FUNCTION_BLOCK FB_LevitationSystem IMPLEMENTS ITF_HighLevelSystem
VAR_INPUT
	eState : LevitationSystemSTM;
	nTGControlOption : USINT;
	eActivationStatus : ActivationStatus;
END_VAR
VAR_OUTPUT
	bEnableCurrentController : BOOL;
	bEnableIControl : BOOL;
	bEnablePControl : BOOL;
END_VAR
VAR
	fbEqualizingControl			: FB_EqualizingController;
	fbTrajectoryGeneratorXMC1	: FB_TrajectoryGenerator;
	fbTrajectoryGeneratorXMC2	: FB_TrajectoryGenerator;
	fbTrajectoryGeneratorXMC3	: FB_TrajectoryGenerator;
	fbTrajectoryGeneratorXMC4	: FB_TrajectoryGenerator;
	
	fActualLevDistanceForFmag : ARRAY [0..3] OF REAL;
	fActualLevCurrentForFmag : ARRAY [0..3] OF REAL;
END_VAR

IF eActivationStatus = ActivationStatus.Enabled THEN
	//High Level State Machine
	CASE eState OF
		LevitationSystemSTM.Idling:
			;
			
			
		LevitationSystemSTM.Stationary:
			bEnableCurrentController := FALSE;
			fbTrajectoryGeneratorXMC1.bTransition := FALSE;
			fbTrajectoryGeneratorXMC2.bTransition := FALSE;
			fbTrajectoryGeneratorXMC3.bTransition := FALSE;
			fbTrajectoryGeneratorXMC4.bTransition := FALSE;

			fbEqualizingControl.bActive := FALSE;		
		
			doSetOperationMode();
			
			fbTrajectoryGeneratorXMC1();
			fbTrajectoryGeneratorXMC2();
			fbTrajectoryGeneratorXMC3();
			fbTrajectoryGeneratorXMC4();
			fbEqualizingControl();
			
		LevitationSystemSTM.Transitioning:
			bEnableCurrentController := TRUE;
			fbTrajectoryGeneratorXMC1.bTransition := TRUE;
			fbTrajectoryGeneratorXMC2.bTransition := TRUE;
			fbTrajectoryGeneratorXMC3.bTransition := TRUE;
			fbTrajectoryGeneratorXMC4.bTransition := TRUE;
			
			fbEqualizingControl.bActive := FALSE;
			
			fbTrajectoryGeneratorXMC1();
			fbTrajectoryGeneratorXMC2();
			fbTrajectoryGeneratorXMC3();
			fbTrajectoryGeneratorXMC4();
			fbEqualizingControl();
			
			
		LevitationSystemSTM.HoldingAirGap:
			bEnableCurrentController := FALSE;
			fbTrajectoryGeneratorXMC1.bTransition := FALSE;
			fbTrajectoryGeneratorXMC2.bTransition := FALSE;
			fbTrajectoryGeneratorXMC3.bTransition := FALSE;
			fbTrajectoryGeneratorXMC4.bTransition := FALSE;
			
			fbEqualizingControl.bActive := TRUE;
			
			doCalculateFmagValuesForEC(	fActualLevDistance := fActualLevDistanceForFmag,			//to be implemented
										fActualCurrent := fActualLevCurrentForFmag);
			
			fbTrajectoryGeneratorXMC1();
			fbTrajectoryGeneratorXMC2();
			fbTrajectoryGeneratorXMC3();
			fbTrajectoryGeneratorXMC4();
			fbEqualizingControl();
			
			
		LevitationSystemSTM.TransitioningToZero:
			bEnableCurrentController := TRUE;
			fbTrajectoryGeneratorXMC1.bTransition := TRUE;
			fbTrajectoryGeneratorXMC2.bTransition := TRUE;
			fbTrajectoryGeneratorXMC3.bTransition := TRUE;
			fbTrajectoryGeneratorXMC4.bTransition := TRUE;
			
			fbEqualizingControl.bActive := FALSE;
			
			doSetPresetTGValuesForBackToGround();		//to be implemented with Controller structure
			
			fbTrajectoryGeneratorXMC1();
			fbTrajectoryGeneratorXMC2();
			fbTrajectoryGeneratorXMC3();
			fbTrajectoryGeneratorXMC4();
			fbEqualizingControl();
			
	END_CASE	

END_IF

PROPERTY PUBLIC aECOutputZVector : ARRAY [0..3] OF REAL
GET
END_GET
END_PROPERTY

PROPERTY PUBLIC aTGActualLevAcceleration : ARRAY [0..3] OF REAL
SET
END_SET
END_PROPERTY

PROPERTY PUBLIC aTGActualLevCurrent : ARRAY [0..3] OF REAL
SET
fActualLevCurrentForFmag := aTGActualLevCurrent;
END_SET
END_PROPERTY

PROPERTY PUBLIC aTGActualLevDistance : ARRAY [0..3] OF REAL
SET
fActualLevDistanceForFmag := aTGActualLevDistance;
END_SET
END_PROPERTY

PROPERTY PUBLIC aTGActualLevVelocity : ARRAY [0..3] OF REAL
SET
END_SET
END_PROPERTY

PROPERTY PUBLIC aTGOutputLevAcceleration : ARRAY [0..3] OF REAL
GET
END_GET
END_PROPERTY

PROPERTY PUBLIC aTGOutputLevCurrent : ARRAY [0..3] OF REAL
GET
END_GET
END_PROPERTY

PROPERTY PUBLIC aTGOutputLevDistance : ARRAY [0..3] OF REAL
GET
END_GET
END_PROPERTY

PROPERTY PUBLIC aTGOutputLevForce : ARRAY [0..3] OF REAL
GET
END_GET
END_PROPERTY

PROPERTY PUBLIC aTGOutputLevVelocity : ARRAY [0..3] OF REAL
GET
END_GET
END_PROPERTY

PROPERTY PUBLIC aTGOutputLevVoltage : ARRAY [0..3] OF REAL
GET
END_GET
END_PROPERTY

PROPERTY PUBLIC bTrajectoryCompleted : BOOL
GET
VAR
	bTrajectoryCompletedXMC1 : BOOL;
	bTrajectoryCompletedXMC2 : BOOL;
	bTrajectoryCompletedXMC3 : BOOL;
	bTrajectoryCompletedXMC4 : BOOL;
END_VAR
bTrajectoryCompletedXMC1 := fbTrajectoryGeneratorXMC1.bTrajectoryCompleted;
bTrajectoryCompletedXMC2 := fbTrajectoryGeneratorXMC2.bTrajectoryCompleted;
bTrajectoryCompletedXMC3 := fbTrajectoryGeneratorXMC3.bTrajectoryCompleted;
bTrajectoryCompletedXMC4 := fbTrajectoryGeneratorXMC4.bTrajectoryCompleted;

IF bTrajectoryCompletedXMC1 AND bTrajectoryCompletedXMC2 AND bTrajectoryCompletedXMC3 AND bTrajectoryCompletedXMC4 THEN
	bTrajectoryCompleted := TRUE;
ELSE
	bTrajectoryCompleted := FALSE;
END_IF
END_GET
SET
END_SET
END_PROPERTY

METHOD PRIVATE doCalculateFmagValuesForEC
VAR_INPUT
	fActualLevDistance : ARRAY [0..3] OF REAL;
	fActualCurrent		: ARRAY [0..3] OF REAL;
END_VAR
fbEqualizingControl.fActualDeltaFmag := 0;
END_METHOD

METHOD PRIVATE doSetOperationMode
VAR_INPUT
END_VAR
IF nTGControlOption.0 THEN
	fbTrajectoryGeneratorXMC1.eMode := TGControllerMode.IControl;
	fbTrajectoryGeneratorXMC2.eMode := TGControllerMode.IControl;
	fbTrajectoryGeneratorXMC3.eMode := TGControllerMode.IControl;
	fbTrajectoryGeneratorXMC4.eMode := TGControllerMode.IControl;
	
	bEnableIControl := TRUE;
	bEnablePControl := FALSE;
END_IF

IF nTGControlOption.1 THEN
	fbTrajectoryGeneratorXMC1.eMode := TGControllerMode.PControl;
	fbTrajectoryGeneratorXMC2.eMode := TGControllerMode.PControl;
	fbTrajectoryGeneratorXMC3.eMode := TGControllerMode.PControl;
	fbTrajectoryGeneratorXMC4.eMode := TGControllerMode.PControl;
	
	bEnableIControl := FALSE;
	bEnablePControl := TRUE;
END_IF
END_METHOD

METHOD PRIVATE doSetPresetTGValuesForBackToGround
VAR_INPUT
END_VAR
END_METHOD

PROPERTY eCondition : HighLevelCondition
GET
IF eActivationStatus = ActivationStatus.Disabled THEN
	eCondition := HighLevelCondition.SLEEP;
ELSE
	IF fbTrajectoryGeneratorXMC1.eCondition = SubLevelCondition.RUN AND fbTrajectoryGeneratorXMC2.eCondition = SubLevelCondition.RUN AND fbTrajectoryGeneratorXMC3.eCondition = SubLevelCondition.RUN AND fbTrajectoryGeneratorXMC4.eCondition = SubLevelCondition.RUN AND fbEqualizingControl.eCondition = SubLevelCondition.RUN THEN
		eCondition := HighLevelCondition.RUN;
	ELSE
		eCondition := HighLevelCondition.INIT;
	END_IF
END_IF
END_GET
END_PROPERTY

PROPERTY PUBLIC fTGDesiredLevAcceleration : REAL
SET
END_SET
END_PROPERTY

PROPERTY PUBLIC fTGDesiredLevDistance : REAL
SET
END_SET
END_PROPERTY

PROPERTY PUBLIC fTGDesiredLevTime : REAL
SET
END_SET
END_PROPERTY

PROPERTY PUBLIC fTGDesiredLevVelocity : REAL
SET
END_SET
END_PROPERTY

PROPERTY nErrorID : UDINT
GET
VAR
	nErrorBitsTG1 : UDINT;
	nErrorBitsTG2 : UDINT;
	nErrorBitsTG3 : UDINT;
	nErrorBitsTG4 : UDINT;
	nErrorBitsEC	: UDINT;
END_VAR
nErrorBitsTG1 := fbTrajectoryGeneratorXMC1.nErrorID;
nErrorBitsTG2 := fbTrajectoryGeneratorXMC2.nErrorID;
nErrorBitsTG3 := fbTrajectoryGeneratorXMC3.nErrorID;
nErrorBitsTG4 := fbTrajectoryGeneratorXMC4.nErrorID;
nErrorBitsEC := fbEqualizingControl.nErrorID;


nErrorID.0 := nErrorBitsEC.0;
nErrorID.1 := nErrorBitsEC.1;
nErrorID.2 := nErrorBitsTG1.0;
nErrorID.3 := nErrorBitsTG1.1;
nErrorID.4 := nErrorBitsTG1.2;
nErrorID.5 := nErrorBitsTG1.3;
nErrorID.6 := nErrorBitsTG1.4;
nErrorID.7 := nErrorBitsTG1.5;
nErrorID.8 := nErrorBitsTG2.0;
nErrorID.9 := nErrorBitsTG2.1;
nErrorID.10 := nErrorBitsTG2.2;
nErrorID.11 := nErrorBitsTG2.3;
nErrorID.12 := nErrorBitsTG2.4;
nErrorID.13 := nErrorBitsTG2.5;
nErrorID.14 := nErrorBitsTG3.0;
nErrorID.15 := nErrorBitsTG3.1;
nErrorID.16 := nErrorBitsTG3.2;
nErrorID.17 := nErrorBitsTG3.3;
nErrorID.18 := nErrorBitsTG3.4;
nErrorID.19 := nErrorBitsTG3.5;
nErrorID.20 := nErrorBitsTG4.0;
nErrorID.21 := nErrorBitsTG4.1;
nErrorID.22 := nErrorBitsTG4.2;
nErrorID.23 := nErrorBitsTG4.3;
nErrorID.24 := nErrorBitsTG4.4;
nErrorID.25 := nErrorBitsTG4.5;
END_GET
END_PROPERTY

END_FUNCTION_BLOCK

(* stored: Version 1.1.0.1, ProductVersion 3.1.4024.12
   POU FB_LevitationSystem: Id {62be560f-4773-4be3-a5a8-e6fcaa9fdc5e}, SpecialFunc None
   Property aECOutputZVector: Id {e8532ec2-c741-4b7b-8b34-a86b44b03236}
   Get Get: Id {2886c540-a581-41eb-8c41-547e16ec48e4}
   Property aTGActualLevAcceleration: Id {223323b8-5081-4179-94ac-03d2f14d212b}
   Set Set: Id {f676f675-5f6c-4f32-b4c4-e7b1269bc728}
   Property aTGActualLevCurrent: Id {0be7462b-6573-4a02-be7b-93c70a347544}
   Set Set: Id {132d2861-3048-430b-857b-95e8d2935efc}
   Property aTGActualLevDistance: Id {5046c194-c4c2-41f8-a8a8-e78e72a7ded7}
   Set Set: Id {61ed663e-d7d3-40b2-80c2-79b58851bac4}
   Property aTGActualLevVelocity: Id {99a5e28f-d915-4b7f-a983-09fd068b463c}
   Set Set: Id {676cfcdf-1f41-4709-b49d-6ae3ae2112c3}
   Property aTGOutputLevAcceleration: Id {9ff96936-9d92-4742-abdd-c6e2b715dfde}
   Get Get: Id {609f8081-1b06-494e-8cf3-373463df83c1}
   Property aTGOutputLevCurrent: Id {749215b4-0f25-4f3a-a13e-6b0f9e0bc0db}
   Get Get: Id {3926eec6-ff0d-4850-9e8b-8f4721874900}
   Property aTGOutputLevDistance: Id {a525620f-a95c-4310-9ef4-b0706473d2dd}
   Get Get: Id {3f50377b-baf2-4b15-a593-ac09cb9accd1}
   Property aTGOutputLevForce: Id {2edc9ced-0973-4a0f-b84f-0f8c31152fde}
   Get Get: Id {98ec0235-6da3-4c91-a90d-c02da730a3da}
   Property aTGOutputLevVelocity: Id {3c1275c5-baab-44c5-80b7-7cd712ea869d}
   Get Get: Id {b99a3ab7-405d-46c8-9f7d-bd439061c6ee}
   Property aTGOutputLevVoltage: Id {b58819ab-83fe-4f1f-80fa-54ccace675d6}
   Get Get: Id {b1fb6c7c-e8ca-41d6-96e3-9cd73edc1693}
   Property bTrajectoryCompleted: Id {9ef7b94f-3f1b-49c8-a2d6-5d9ceff37f18}
   Get Get: Id {5f45c12e-ba03-4b17-a7ef-cf1d1da31a42}
   Set Set: Id {5d4fde02-7326-40bb-a5d9-c86bedd74173}
   Method doCalculateFmagValuesForEC: Id {e883aacb-677e-4abe-ae24-fd1b7b2de366}
   Method doSetOperationMode: Id {04abb227-7b23-46c2-a2f2-c815e00ae789}
   Method doSetPresetTGValuesForBackToGround: Id {9ef85455-36d9-41a4-9ec5-09b3d4f02c32}
   Property eCondition: Id {01bd39e6-00b0-4a87-b944-8315fa4050a7}
   Get Get: Id {eabfe548-b26e-444c-9a2c-8dd71b94c621}
   Property fTGDesiredLevAcceleration: Id {c6c0ecad-e32b-4ac9-b8a8-a8279cf4720d}
   Set Set: Id {b95cf893-e7a9-4b53-967d-79cdcb7aebb0}
   Property fTGDesiredLevDistance: Id {a6febd5f-3b05-4eb1-9d9d-5e4337d07380}
   Set Set: Id {fc744593-7ca5-461c-a06d-5180702e0bb4}
   Property fTGDesiredLevTime: Id {6d90bcae-d970-4748-8bfb-dfd813e9b1d1}
   Set Set: Id {b09ee043-50b8-42f4-91a1-a1ca1123d64b}
   Property fTGDesiredLevVelocity: Id {8c6cc0bf-9f9b-48ea-a429-1827f8b47d30}
   Set Set: Id {86213a2a-051b-4fe4-a239-c088a9b8c020}
   Property nErrorID: Id {139cbef2-6b76-4dea-9e3e-a0544066e7ca}
   Get Get: Id {551a494a-7956-4b5e-8fe2-d72ed847ef0c} *)
